PROGRAM PRG_Cintas
VAR
END_VAR


(* Dependiendo de las detecciones de los sensores, se activarán según qué líneas*)

IF NOT PRG_PickAndPlace.CajaLlenaA THEN
	IF GVL_ProcesoPallet.iLightArrayEmitterA THEN
		GVL_ProcesoPallet.sRollerConveyor.bRollerAzul1 := FALSE;
	ELSE
		GVL_ProcesoPallet.sRollerConveyor.bRollerAzul1 := TRUE;
	END_IF
END_IF

IF NOT PRG_PickAndPlace.CajaLlenaV THEN
	IF GVL_ProcesoPallet.iLightArrayEmitterV THEN
		GVL_ProcesoPallet.sRollerConveyor.bRollerVerde1 := FALSE;
	ELSE
		GVL_ProcesoPallet.sRollerConveyor.bRollerVerde1 := TRUE;
	END_IF
END_IF

IF NOT PRG_PickAndPlace.CajaLlenaM THEN
	IF GVL_ProcesoPallet.iLightArrayEmitterM THEN
		GVL_ProcesoPallet.sRollerConveyor.bRollerMetal1 := FALSE;
	ELSE
		GVL_ProcesoPallet.sRollerConveyor.bRollerMetal1 := TRUE;
	END_IF
END_IF

END_PROGRAM

(* stored: Version 1.1.0.1, ProductVersion 3.1.4024.12
   POU PRG_Cintas: Id {13bfe8b4-6369-4a2c-ac5e-5e576921d46e}, SpecialFunc None *)
